FUNCTION_BLOCK FB_System_BelHa_Sensorik
VAR_INPUT
END_VAR
VAR_OUTPUT
	(* Helligkeit Sensor 1*)
	HelligkeitSensor_1_OUT	: REAL;
	HelligkeitSensor_2_OUT	: REAL;
	(* Helligkeit Sensor 2*)
END_VAR
VAR
	(* Hardware oder DALI *)
	SensorHalle1				: FB_Bel_Lichtsensor;
	HelligkeitSensor_1_IN		: REAL;
	HelligkeitSensor_2_IN		: REAL;
END_VAR

(* ggfs Umrechung *)
HelligkeitSensor_1_OUT := HelligkeitSensor_1_IN * 3 ;
HelligkeitSensor_2_OUT := HelligkeitSensor_2_IN * 3;

END_FUNCTION_BLOCK

(* stored: Version 1.1.0.1, ProductVersion 3.1.4024.9
   POU FB_System_BelHa_Sensorik: Id {bbe167d5-f73e-45b1-afd3-42c2dd49a4fb}, SpecialFunc None *)
